(* CoDeSys 2.3.9.37 project: CapB_1.pro *)
(* Libraries: Standard.lib 4.10.05 12:14:46 *)

(* POU PLC_PRG, ST *)
PROGRAM PLC_PRG
VAR
  Alarma:BOOL;
  posx:INT:=0;
  posy:INT:=0;
  angulo:INT:=0;
  escala:REAL:=1000;
	subex: BOOL;
	bajax: BOOL;
	subey: BOOL;
	bajay: BOOL;
	subeang: BOOL;
	bajaang: BOOL;
	subeesc: BOOL;
	bajaesc: BOOL;
END_VAR
CambiaLetra();

IF subex THEN
    posx:=posx+1;
END_IF


IF bajax THEN
    posx:=posx-1;
END_IF


IF subey THEN
    posy:=posy+1;
END_IF


IF bajay THEN
    posy:=posy-1;
END_IF



IF subeesc THEN
    escala:=escala+10;
END_IF


IF bajaesc THEN
    escala:=escala-10;
END_IF


IF subeang THEN
    angulo:=angulo+1;
END_IF


IF bajaang THEN
    angulo:=angulo-1;
END_IF
END_PROGRAM

(* POU CambiaLetra, ST *)
PROGRAM CambiaLetra
VAR
	M: BOOL;
	ColorLetra: DWORD;
       AlturaLetra:INT;
END_VAR
IF M THEN
  AlturaLetra:=16;
  ColorLetra:=16#FF00FF;
ELSE
   AlturaLetra:=22;
 ColorLetra:=16#121212;
END_IF
END_PROGRAM

(* Visualisation EjemploVisu
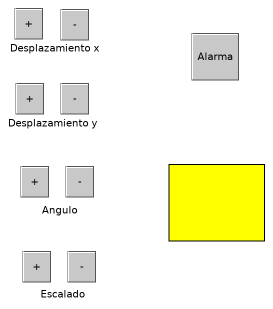
button at (334,35)-(362,66): text "+"; taps PLC_PRG.subex
button at (380,36)-(408,67): text "-"; taps PLC_PRG.bajax
rectangle at (488,191)-(584,268): alarm colour if PLC_PRG.Alarma; x offset PLC_PRG.posx; y offset PLC_PRG.posy; scale PLC_PRG.escala; angle PLC_PRG.angulo
button at (335,110)-(363,141): text "+"; taps PLC_PRG.subey
button at (380,110)-(408,141): text "-"; taps PLC_PRG.bajay
button at (340,193)-(368,224): text "+"; taps PLC_PRG.subeang
button at (385,193)-(413,224): text "-"; taps PLC_PRG.bajaang
button at (342,278)-(370,309): text "+"; taps PLC_PRG.subeesc
button at (387,278)-(415,309): text "-"; taps PLC_PRG.bajaesc
rectangle at (305,60)-(443,90): text "Desplazamiento x"
rectangle at (303,135)-(441,165): text "Desplazamiento y"
rectangle at (310,222)-(448,252): text "Angulo"
rectangle at (313,306)-(451,336): text "Escalado"
button at (511,60)-(558,107): text "Alarma"; toggles PLC_PRG.Alarma
1 elements of other kinds (tables, trends, ...) not read
*)
